FUNCTION F_Decoder : LREAL
VAR_INPUT
		// encoder steps
	input :	ULINT;
	// phase in degrees
	phase : LREAL := 0.0;
	// encoder full turn
	modulus : LREAL := 262144.0;
END_VAR
VAR
	degrees: LREAL;
END_VAR

degrees := 360.0 * ULINT_TO_LREAL(input) / modulus - phase;
IF degrees > 180.0 THEN
	F_Decoder := degrees - 360.0;
ELSE
	F_Decoder := degrees;
END_IF

END_FUNCTION

(* stored: Version 1.1.0.1, ProductVersion 3.1.4024.0
   POU F_Decoder: Id {a3e69684-e86d-4114-aa13-116115eded0c}, SpecialFunc None *)
